{attribute 'qualified_only'}
VAR_GLOBAL
	recipememory: ARRAY [0..1800] OF moveBuffer1kms;
END_VAR

(* stored: Version 1.1.0.1, ProductVersion 3.1.4024.3
   GVL RecipeData: Id {c5e507d1-e960-4d5e-81a0-ba0c9e573e6a} *)
